Universal Robots PolyScope program: bearing_v1.urp

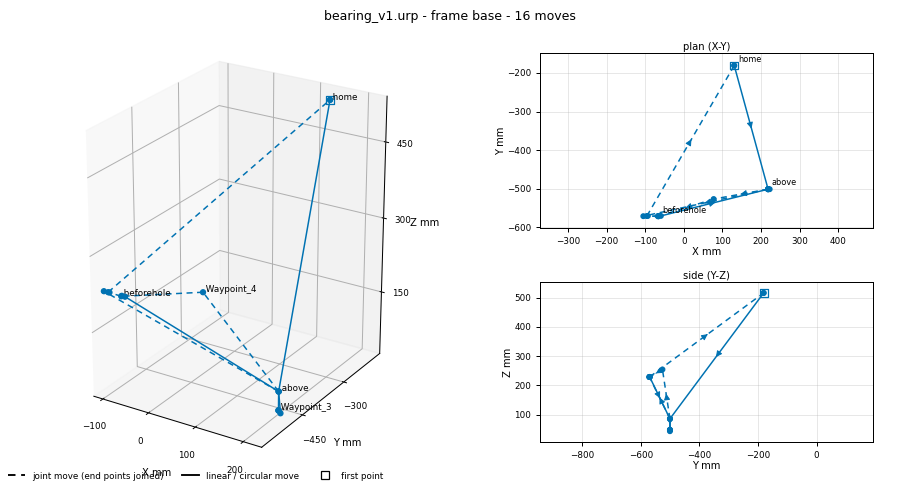
[picture p0: tool path of bearing_v1.urp in frame base, 16 of 25 moves have a stored position in this frame; points joined in program order, loops and branches not executed]
Program bearing_v1 (installation=default directory=/programs/wrs2020 createdIn=5.7.0.90932 lastSavedIn=5.7.0.90932 robotSerialNumber=20205500607)
Calibrated DH parameters: a=[0.000096, -0.337, -0.383372, 0.000118, 0.000015, 0]; d=[0.162724, 79.377998, -95.545185, 16.300583, 0.099689, 0.099499]; alpha=[1.569249, 0.003272, 0.005201, 1.570041, -1.570219, 0]; deltaTheta=[0, 0.65664, 5.410619, 0.215927, -0.000001, 0]
Robot Program (runOnlyOnce=true)
  MoveJ speed 180 deg/s, acceleration 80 deg/s^2 (useActiveTCP=true) feature=Base
    Waypoint home: TCP in base x=130.635 y=-180.692 z=515.97 mm, rx=-0.0117 ry=-3.1402 rz=-0.0315 rad; joints [89.951, -120.324, 80.212, -48.705, -89.957, -0.002] deg; TCP offset x=0 y=0 z=165 mm, rx=0 ry=0 rz=0 rad
  URCap Gripper (Robotiq_Grippers, Robotiq Inc.) dataModel(position=0.0, force=100.0, speed=100.0, positionInDouble=0.0, forceInDouble=100.0, speedInDouble=100.0, slaveIds=[9], blocking=true)
  MoveL speed 250 mm/s, acceleration 1200 mm/s^2 (useActiveTCP=false) tcp=gripper_85_tip; feature=Base
    Waypoint above: TCP in base x=218.287 y=-500.902 z=86.011 mm, rx=-2.1841 ry=2.228 rz=-0.024 rad; joints [98.796, -75.562, 110.256, -124.664, -88.151, -80.024] deg
    Waypoint Waypoint_3: TCP in base x=218.287 y=-500.902 z=48.168 mm, rx=-2.1841 ry=2.228 rz=-0.024 rad; joints [98.784, -72.218, 112.615, -130.368, -88.157, -80] deg; TCP offset x=0 y=0 z=165 mm, rx=0 ry=0 rz=0 rad
  URCap Gripper (Robotiq_Grippers, Robotiq Inc.) dataModel(position=100.0, force=0.0, speed=0.0, positionInDouble=100.0, forceInDouble=0.0, speedInDouble=0.0, slaveIds=[9], blocking=true)
  URCap Gripper (Robotiq_Grippers, Robotiq Inc.) dataModel(position=0.0, force=0.0, speed=0.0, positionInDouble=0.0, forceInDouble=0.0, speedInDouble=0.0, slaveIds=[9], blocking=true)
  MoveL speed 600 mm/s, acceleration 1200 mm/s^2 (useActiveTCP=false) tcp=gripper_85_tip; feature=Base
    Waypoint Waypoint_2: TCP in base x=218.287 y=-500.902 z=48.168 mm, rx=-0.0072 ry=3.1154 rz=0.0062 rad; joints [98.784, -72.218, 112.615, -130.368, -88.157, 8.595] deg; TCP offset x=0 y=0 z=165 mm, rx=0 ry=0 rz=0 rad
  URCap Gripper (Robotiq_Grippers, Robotiq Inc.) dataModel(position=100.0, force=0.0, speed=0.0, positionInDouble=100.0, forceInDouble=0.0, speedInDouble=0.0, slaveIds=[9], blocking=true)
  URCap Gripper (Robotiq_Grippers, Robotiq Inc.) dataModel(position=14.117647058823529, force=0.0, speed=0.0, positionInDouble=14.117647058823529, forceInDouble=0.0, speedInDouble=0.0, slaveIds=[9], blocking=true)
  MoveL speed 600 mm/s, acceleration 1200 mm/s^2 (useActiveTCP=false) tcp=gripper_85_tip; feature=Base
    Waypoint Waypoint_3: TCP in base x=218.287 y=-500.902 z=48.168 mm, rx=-2.1841 ry=2.228 rz=-0.024 rad; joints [98.784, -72.218, 112.615, -130.368, -88.157, -80] deg; TCP offset x=0 y=0 z=165 mm, rx=0 ry=0 rz=0 rad
    Waypoint Waypoint_1: TCP in base x=222.423 y=-500.902 z=43.626 mm, rx=-1.9097 ry=1.9461 rz=-0.5001 rad; joints [85.342, -72.496, 119.915, -134.531, -60.23, -94.253] deg; TCP offset x=0 y=0 z=165 mm, rx=0 ry=0 rz=0 rad
  URCap Gripper (Robotiq_Grippers, Robotiq Inc.) dataModel(position=100.0, force=100.0, speed=100.0, positionInDouble=100.0, forceInDouble=100.0, speedInDouble=100.0, slaveIds=[9], blocking=true)
  MoveL speed 250 mm/s, acceleration 1200 mm/s^2 (useActiveTCP=false) tcp=gripper_85_tip; feature=Base
    Waypoint above: TCP in base x=218.287 y=-500.902 z=86.011 mm, rx=-2.1841 ry=2.228 rz=-0.024 rad; joints [98.796, -75.562, 110.256, -124.664, -88.151, -80.024] deg
  SuppressedNode
    MoveJ speed 60 deg/s, acceleration 80 deg/s^2 (useActiveTCP=true) feature=Base
      Waypoint intermediate: motionParameters(blendRadius=0.05); TCP in base x=115.537 y=-464.392 z=278.491 mm, rx=2.1151 ry=-1.8246 rz=-0.1767 rad; joints [98.791, -95.537, 106.25, -108.287, -109.219, -91.027] deg
      Waypoint before_hole: TCP in base x=-57.686 y=-570.408 z=232.23 mm, rx=1.3727 ry=-1.1616 rz=-1.3181 rad; joints [97.319, -59.573, 88.654, -50.464, -171.504, -31.295] deg
  SuppressedNode
    MoveJ speed 60 deg/s, acceleration 80 deg/s^2 (useActiveTCP=true) feature=Base
      Waypoint at_hole: TCP in base x=-85.495 y=-570.408 z=232.23 mm, rx=1.3727 ry=-1.1616 rz=-1.3181 rad; joints [94.632, -61.815, 93.453, -62.169, -173.913, -40.501] deg; TCP offset x=0 y=0 z=165 mm, rx=0 ry=0 rz=0 rad
  SuppressedNode
    Force Frame feature=Joint_6_name; selection=[0, 0, 1, 0, 0, 0]; wrench=[0, 0, 10, 0, 0, 0]; limitsForce=[0.15, 0.15, 0.01, 1.047198, 1.047198, 1.047198]; limitsMotion=[0.1, 0.1, 0.1, 0.349066, 0.349066, 0.349066]
      MoveJ speed 60 deg/s, acceleration 80 deg/s^2 (useActiveTCP=true) feature=Base
        Waypoint turn_right (Relative): relativeFromPosition TCP in base x=-85.515 y=-570.41 z=232.207 mm, rx=1.3727 ry=-1.1616 rz=-1.3181 rad; joints [94.63, -61.813, 93.454, -62.171, -173.913, -40.501] deg; TCP offset x=0 y=0 z=165 mm, rx=0 ry=0 rz=0 rad; TCP in base x=-85.507 y=-570.407 z=232.241 mm, rx=0.846 ry=-1.441 rz=-0.7763 rad; joints [94.699, -63.491, 97.916, -73.842, -175.626, -8.792] deg
        Waypoint turn_left (Relative): relativeFromPosition TCP in base x=-85.52 y=-570.402 z=232.224 mm, rx=0.846 ry=-1.4411 rz=-0.7763 rad; joints [94.698, -63.49, 97.916, -73.843, -175.624, -8.792] deg; TCP in base x=-85.509 y=-570.398 z=232.173 mm, rx=1.3728 ry=-1.1615 rz=-1.3182 rad; joints [94.631, -61.811, 93.456, -62.169, -173.913, -40.501] deg
        Waypoint turn_left (Relative): relativeFromPosition TCP in base x=-85.52 y=-570.402 z=232.224 mm, rx=0.846 ry=-1.4411 rz=-0.7763 rad; joints [94.698, -63.49, 97.916, -73.843, -175.624, -8.792] deg; TCP in base x=-85.509 y=-570.398 z=232.173 mm, rx=1.3728 ry=-1.1615 rz=-1.3182 rad; joints [94.631, -61.811, 93.456, -62.169, -173.913, -40.501] deg
        Waypoint turn_right (Relative): relativeFromPosition TCP in base x=-85.515 y=-570.41 z=232.207 mm, rx=1.3727 ry=-1.1616 rz=-1.3181 rad; joints [94.63, -61.813, 93.454, -62.171, -173.913, -40.501] deg; TCP in base x=-85.507 y=-570.407 z=232.241 mm, rx=0.846 ry=-1.441 rz=-0.7763 rad; joints [94.699, -63.491, 97.916, -73.842, -175.626, -8.792] deg
  MoveJ speed 60 deg/s, acceleration 80 deg/s^2 (useActiveTCP=false) tcp=gripper_85_tip; feature=Base
    Waypoint Waypoint_4: motionParameters(blendRadius=0.05); TCP in base x=77.346 y=-526.445 z=254.497 mm, rx=2.1138 ry=-1.9338 rz=-0.2706 rad; joints [93.109, -85.443, 98.102, -105.695, -107.975, -92.542] deg
    Waypoint beforehole: TCP in base x=-66.725 y=-571.237 z=228.439 mm, rx=1.497 ry=-1.6176 rz=-0.8285 rad; joints [93.116, -71.584, 102.92, -120.139, -149.991, -81.706] deg
  MoveJ speed 60 deg/s, acceleration 80 deg/s^2 (useActiveTCP=false) tcp=gripper_85_tip; feature=Base
    Waypoint athole: TCP in base x=-93.062 y=-570.055 z=228.956 mm, rx=1.497 ry=-1.6176 rz=-0.8285 rad; joints [90.445, -71.97, 104.758, -126.218, -149.936, -87.03] deg
  Force Frame feature=Base; selection=[1, 1, 1, 0, 0, 0]; wrench=[-10, 0, 0, 0, 0, 0]; limitsForce=[0.01, 0.01, 0.01, 1.047198, 1.047198, 1.047198]; limitsMotion=[0.1, 0.1, 0.1, 0.349066, 0.349066, 0.349066]
    MoveL speed 250 mm/s, acceleration 1200 mm/s^2 (useActiveTCP=false) tcp=gripper_85_tip; feature=Base
      MoveDirectionNode (selectedDirection=YPlus toolParams=0.005, 0.02)
        Until DISTANCE (allowActions=false deceleration=3 distanceNodeType=STOP) Distance=0.001; motionParameters(blendRadius=0)
      MoveDirectionNode (selectedDirection=ZMinus toolParams=0.005, 0.02)
        Until DISTANCE (allowActions=false deceleration=3 distanceNodeType=STOP) Distance=0.001; motionParameters(blendRadius=0)
      MoveDirectionNode (selectedDirection=YMinus toolParams=0.005, 0.02)
        Until DISTANCE (allowActions=false deceleration=3 distanceNodeType=STOP) Distance=0.001; motionParameters(blendRadius=0)
      MoveDirectionNode (selectedDirection=YMinus toolParams=0.005, 0.02)
        Until DISTANCE (allowActions=false deceleration=3 distanceNodeType=STOP) Distance=0.001; motionParameters(blendRadius=0)
      MoveDirectionNode (selectedDirection=ZPlus toolParams=0.005, 0.02)
        Until DISTANCE (allowActions=false deceleration=3 distanceNodeType=STOP) Distance=0.001; motionParameters(blendRadius=0)
      MoveDirectionNode (selectedDirection=YPlus toolParams=0.005, 0.02)
        Until DISTANCE (allowActions=false deceleration=3 distanceNodeType=STOP) Distance=0.001; motionParameters(blendRadius=0)
      MoveDirectionNode (selectedDirection=YPlus toolParams=0.005, 0.02)
        Until DISTANCE (allowActions=false deceleration=3 distanceNodeType=STOP) Distance=0.001; motionParameters(blendRadius=0)
      MoveDirectionNode (selectedDirection=ZPlus toolParams=0.005, 0.02)
        Until DISTANCE (allowActions=false deceleration=3 distanceNodeType=STOP) Distance=0.001; motionParameters(blendRadius=0)
      MoveDirectionNode (selectedDirection=YMinus toolParams=0.005, 0.02)
        Until DISTANCE (allowActions=false deceleration=3 distanceNodeType=STOP) Distance=0.001; motionParameters(blendRadius=0)
      MoveDirectionNode (selectedDirection=YMinus toolParams=0.005, 0.02)
        Until DISTANCE (allowActions=false deceleration=3 distanceNodeType=STOP) Distance=0.001; motionParameters(blendRadius=0)
      MoveDirectionNode (selectedDirection=ZMinus toolParams=0.005, 0.02)
        Until DISTANCE (allowActions=false deceleration=3 distanceNodeType=STOP) Distance=0.001; motionParameters(blendRadius=0)
      MoveDirectionNode (selectedDirection=YPlus toolParams=0.005, 0.02)
        Until DISTANCE (allowActions=false deceleration=3 distanceNodeType=STOP) Distance=0.001; motionParameters(blendRadius=0)
  If pose_dist(get_actual_tcp_pose(), push_1_done) > .005
    Force Frame feature=Base; selection=[1, 0, 0, 0, 0, 0]; wrench=[-10, 0, 10, 0, 0, 0]; limitsForce=[0.01, 0.15, 0.01, 1.047198, 1.047198, 1.047198]; limitsMotion=[0.1, 0.1, 0.1, 0.349066, 0.349066, 0.349066]
      MoveL speed 50 mm/s, acceleration 200 mm/s^2 (useActiveTCP=false) tcp=gripper_85_tip; feature=Base
        Waypoint rightturn (Relative): relativeFromPosition TCP in base x=-93.069 y=-570.049 z=228.937 mm, rx=1.497 ry=-1.6176 rz=-0.8285 rad; joints [90.445, -71.969, 104.759, -126.217, -149.936, -87.029] deg; TCP in base x=-93.056 y=-570.054 z=228.975 mm, rx=1.1857 ry=-1.6671 rz=-0.4357 rad; joints [90.457, -71.686, 115.038, -161.493, -150.211, -86.762] deg
        Waypoint leftturn (Relative): relativeFromPosition TCP in base x=-93.048 y=-570.049 z=228.934 mm, rx=1.1858 ry=-1.6671 rz=-0.4357 rad; joints [90.457, -71.685, 115.04, -161.493, -150.208, -86.762] deg; TCP in base x=-93.069 y=-570.047 z=228.952 mm, rx=1.497 ry=-1.6176 rz=-0.8285 rad; joints [90.445, -71.97, 104.758, -126.214, -149.936, -87.03] deg
        Waypoint leftturn (Relative): relativeFromPosition TCP in base x=-93.048 y=-570.049 z=228.934 mm, rx=1.1858 ry=-1.6671 rz=-0.4357 rad; joints [90.457, -71.685, 115.04, -161.493, -150.208, -86.762] deg; TCP in base x=-93.069 y=-570.047 z=228.952 mm, rx=1.497 ry=-1.6176 rz=-0.8285 rad; joints [90.445, -71.97, 104.758, -126.214, -149.936, -87.03] deg
        Waypoint rightturn (Relative): relativeFromPosition TCP in base x=-93.069 y=-570.049 z=228.937 mm, rx=1.497 ry=-1.6176 rz=-0.8285 rad; joints [90.445, -71.969, 104.759, -126.217, -149.936, -87.029] deg; TCP in base x=-93.056 y=-570.054 z=228.975 mm, rx=1.1857 ry=-1.6671 rz=-0.4357 rad; joints [90.457, -71.686, 115.038, -161.493, -150.211, -86.762] deg
  SuppressedNode
    If pose_dist(get_actual_tcp_pose(), athole) < .005
      Popup Message (haltProgram=false message=bearing insertion seems to have failed inputType=Text)
  URCap Gripper (Robotiq_Grippers, Robotiq Inc.) dataModel(position=0.0, force=0.0, speed=100.0, positionInDouble=0.0, forceInDouble=0.0, speedInDouble=100.0, slaveIds=[9], blocking=true)
  MoveJ speed 60 deg/s, acceleration 80 deg/s^2 (useActiveTCP=false) tcp=gripper_85_tip; feature=Base
    Waypoint Waypoint_6 (Relative): relativeFromPosition TCP in base x=-104.624 y=-570.1 z=229.071 mm, rx=1.4967 ry=-1.6177 rz=-0.8284 rad; joints [89.261, -71.985, 105.381, -128.866, -149.849, -89.368] deg; TCP in base x=-90.708 y=-570.103 z=229.07 mm, rx=1.4967 ry=-1.6177 rz=-0.8284 rad; joints [90.688, -71.962, 104.605, -125.653, -149.956, -86.534] deg
  URCap Gripper (Robotiq_Grippers, Robotiq Inc.) dataModel(position=100.0, force=100.0, speed=100.0, positionInDouble=100.0, forceInDouble=100.0, speedInDouble=100.0, slaveIds=[9], blocking=true)
  If rq_current_pos_mm()<10
    'Gripper fully closed = bearing not inserted!! Stopping.'
    MoveL speed 100 mm/s, acceleration 60 mm/s^2 (useActiveTCP=false) tcp=gripper_85_tip; feature=Base
      MoveDirectionNode (selectedDirection=XPlus) feature=Base
        Until DISTANCE (allowActions=false deceleration=3 distanceNodeType=STOP) Distance=0.1; motionParameters(blendRadius=0)
    Halt
  Force Frame feature=Base; selection=[1, 0, 0, 0, 0, 0]; wrench=[-10, 0, 10, 0, 0, 0]; limitsForce=[0.01, 0.15, 0.01, 1.047198, 1.047198, 1.047198]; limitsMotion=[0.1, 0.1, 0.1, 0.349066, 0.349066, 0.349066]
    MoveL speed 50 mm/s, acceleration 200 mm/s^2 (useActiveTCP=false) tcp=gripper_85_tip; feature=Base
      Waypoint rightturn (Relative): relativeFromPosition TCP in base x=-93.069 y=-570.049 z=228.937 mm, rx=1.497 ry=-1.6176 rz=-0.8285 rad; joints [90.445, -71.969, 104.759, -126.217, -149.936, -87.029] deg; TCP in base x=-93.056 y=-570.054 z=228.975 mm, rx=1.1857 ry=-1.6671 rz=-0.4357 rad; joints [90.457, -71.686, 115.038, -161.493, -150.211, -86.762] deg
      Waypoint leftturn (Relative): relativeFromPosition TCP in base x=-93.048 y=-570.049 z=228.934 mm, rx=1.1858 ry=-1.6671 rz=-0.4357 rad; joints [90.457, -71.685, 115.04, -161.493, -150.208, -86.762] deg; TCP in base x=-93.069 y=-570.047 z=228.952 mm, rx=1.497 ry=-1.6176 rz=-0.8285 rad; joints [90.445, -71.97, 104.758, -126.214, -149.936, -87.03] deg
      Waypoint leftturn (Relative): relativeFromPosition TCP in base x=-93.048 y=-570.049 z=228.934 mm, rx=1.1858 ry=-1.6671 rz=-0.4357 rad; joints [90.457, -71.685, 115.04, -161.493, -150.208, -86.762] deg; TCP in base x=-93.069 y=-570.047 z=228.952 mm, rx=1.497 ry=-1.6176 rz=-0.8285 rad; joints [90.445, -71.97, 104.758, -126.214, -149.936, -87.03] deg
      Waypoint rightturn (Relative): relativeFromPosition TCP in base x=-93.069 y=-570.049 z=228.937 mm, rx=1.497 ry=-1.6176 rz=-0.8285 rad; joints [90.445, -71.969, 104.759, -126.217, -149.936, -87.029] deg; TCP in base x=-93.056 y=-570.054 z=228.975 mm, rx=1.1857 ry=-1.6671 rz=-0.4357 rad; joints [90.457, -71.686, 115.038, -161.493, -150.211, -86.762] deg
  URCap Gripper (Robotiq_Grippers, Robotiq Inc.) dataModel(position=0.0, force=0.0, speed=100.0, positionInDouble=0.0, forceInDouble=0.0, speedInDouble=100.0, slaveIds=[9], blocking=true)
  MoveJ speed 60 deg/s, acceleration 80 deg/s^2 (useActiveTCP=false) tcp=gripper_85_tip; feature=Base
    Waypoint Waypoint_7: TCP in base x=-66.41 y=-570.102 z=229.085 mm, rx=1.4967 ry=-1.6176 rz=-0.8284 rad; joints [93.156, -71.758, 103.037, -120.015, -149.998, -81.615] deg
  URCap Gripper (Robotiq_Grippers, Robotiq Inc.) dataModel(position=100.0, force=100.0, speed=100.0, positionInDouble=100.0, forceInDouble=100.0, speedInDouble=100.0, slaveIds=[9], blocking=true)
  Force Frame feature=Base; selection=[1, 0, 0, 0, 0, 0]; wrench=[-5, 0, 10, 0, 0, 0]; limitsForce=[0.01, 0.15, 0.01, 1.047198, 1.047198, 1.047198]; limitsMotion=[0.1, 0.1, 0.1, 0.349066, 0.349066, 0.349066]
    Wait Sleep waitTime=5
    MoveL speed 5 mm/s, acceleration 5 mm/s^2 (useActiveTCP=false) tcp=gripper_85_tip; feature=Base
      MoveDirectionNode (selectedDirection=XPlus) feature=Joint_6_name
        Until DISTANCE (allowActions=false deceleration=3 distanceNodeType=STOP) Distance=0.0005; motionParameters(blendRadius=0)
    Loop Counting (count=12) loopVariable(name=Loop_2)
      If pose_dist(get_actual_tcp_pose(), push_3_done) > .005
        MoveL speed 5 mm/s, acceleration 5 mm/s^2 (useActiveTCP=false) tcp=gripper_85_tip; feature=Base
          MoveDirectionNode (toolParams=0.005, 0.02) expression=[sin((Loop_2-1)/6*3.141),0.0,-cos((Loop_2-1)/6*3.141)]; feature=Joint_6_name
            Until DISTANCE (allowActions=false deceleration=3 distanceNodeType=STOP) Distance=0.0005; motionParameters(blendRadius=0)
  MoveJ speed 60 deg/s, acceleration 80 deg/s^2 (useActiveTCP=false) tcp=gripper_85_tip; feature=Base
    Waypoint a_bit_back: TCP in base x=-59.374 y=-570.102 z=229.085 mm, rx=1.4967 ry=-1.6176 rz=-0.8284 rad; joints [93.865, -71.658, 102.534, -118.385, -149.976, -80.204] deg
  MoveL speed 250 mm/s, acceleration 1200 mm/s^2 (useActiveTCP=false) tcp=gripper_85_tip; feature=Base
    Waypoint above: TCP in base x=218.287 y=-500.902 z=86.011 mm, rx=-2.1841 ry=2.228 rz=-0.024 rad; joints [98.796, -75.562, 110.256, -124.664, -88.151, -80.024] deg
  If False
    MoveJ speed 60 deg/s, acceleration 80 deg/s^2 (useActiveTCP=false) tcp=gripper_85_tip; feature=Base
      Waypoint push_1_done referenceName=push_1_done: TCP in base x=-104.765 y=-570.8 z=228.861 mm, rx=1.4972 ry=-1.6175 rz=-0.8279 rad; joints [89.242, -71.9, 105.308, -128.958, -149.825, -89.455] deg
      SuppressedNode
        Waypoint Waypoint_5: 
      Waypoint push_3_done referenceName=push_3_done: TCP in base x=-95.643 y=-570.475 z=229.043 mm, rx=1.4967 ry=-1.6178 rz=-0.8287 rad; joints [90.182, -71.929, 104.818, -126.745, -149.925, -87.518] deg
  MoveJ speed 180 deg/s, acceleration 80 deg/s^2 (useActiveTCP=true) feature=Base
    Waypoint home: TCP in base x=130.635 y=-180.692 z=515.97 mm, rx=-0.0117 ry=-3.1402 rz=-0.0315 rad; joints [89.951, -120.324, 80.212, -48.705, -89.957, -0.002] deg
